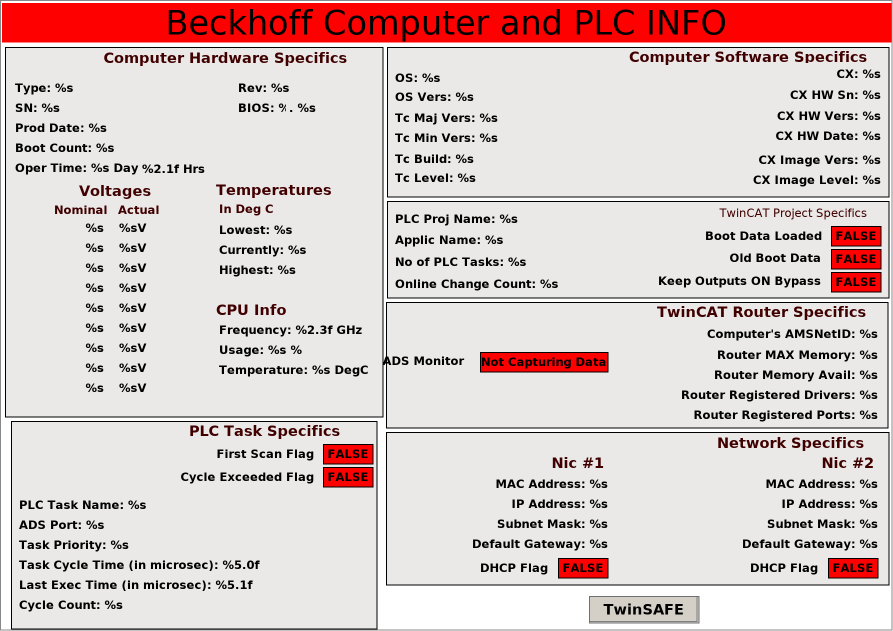
VISUALIZATION TwinCAT_INFO  // 893x631
    Button (589,596 110x27), "TwinSAFE"
        OnMouseClick: change screen: TwinSAFE
    RoundedRectangle (2,3 889x39), "Beckhoff Computer and PLC INFO"
    RoundedRectangle (387,47 502x150)
    Label (614,44 256x26), "Computer Software Specifics"
    Rectangle (392,67 256x22), "OS: %s", text variable: g_stHMI_DevIdent.strImageOsName
    RoundedRectangle (387,201 502x97)
    Label (695,200 175x26), "TwinCAT Project Specifics"
    RoundedRectangle (386,302 502x126)
    Label (613,299 256x26), "TwinCAT Router Specifics"
    RoundedRectangle (11,421 366x208)
    Label (185,418 158x26), "PLC Task Specifics"
    Rectangle (392,86 208x22), "OS Vers: %s", text variable: g_stHMI_DevIdent.strImageOsVersion
    Rectangle (392,107 119x22), "Tc Maj Vers: %s", text variable: g_stHMI_DevIdent.strTwinCATVersion
    Rectangle (392,127 111x22), "Tc Min Vers: %s", text variable: g_stHMI_DevIdent.strTwinCATRevision
    Rectangle (392,148 111x22), "Tc Build: %s", text variable: g_stHMI_DevIdent.strTwinCATBuild
    Rectangle (392,167 111x22), "Tc Level: %s", text variable: g_stHMI_DevIdent.strTwinCATLevel
    Rectangle (738,63 146x22), "CX: %s", text variable: g_stHMI_DevIdent.strHardwareModel
    Rectangle (726,84 158x22), "CX HW Sn: %s", text variable: g_stHMI_DevIdent.strHardwareSerialNo
    Rectangle (733,105 151x22), "CX HW Vers: %s", text variable: g_stHMI_DevIdent.strHardwareVersion
    Rectangle (737,125 147x22), "CX HW Date: %s", text variable: g_stHMI_DevIdent.strHardwareDate
    Rectangle (725,149 159x22), "CX Image Vers: %s", text variable: g_stHMI_DevIdent.strImageVersion
    Rectangle (625,169 259x22), "CX Image Level: %s", text variable: g_stHMI_DevIdent.strImageLevel
    Rectangle (392,208 283x22), "PLC Proj Name: %s", text variable: g_stHMI_AppInfo.ProjectName
    Rectangle (392,229 359x22), "Applic Name: %s", text variable: g_stHMI_AppInfo.AppName
    Rectangle (392,251 155x22), "No of PLC Tasks: %s", text variable: g_stHMI_AppInfo.TaskCnt
    Rectangle (392,273 191x22), "Online Change Count: %s", text variable: g_stHMI_AppInfo.OnlineChangeCnt
    Group (831,226 50x20)
        Rectangle (0,0 50x20), "TRUE", invisible if: NOT g_stHMI_AppInfo.BootDataLoaded
        Rectangle (0,0 50x20), "FALSE", invisible if: g_stHMI_AppInfo.BootDataLoaded
    Label (705,224 120x24), "Boot Data Loaded"
    Group (831,249 50x20)
        Rectangle (0,0 50x20), "TRUE", invisible if: NOT g_stHMI_AppInfo.OldBootData
        Rectangle (0,0 50x20), "FALSE", invisible if: g_stHMI_AppInfo.OldBootData
    Label (726,246 98x24), "Old Boot Data"
    Group (831,272 50x20)
        Rectangle (0,0 50x20), "TRUE", invisible if: NOT g_stHMI_AppInfo.KeepOutputsOnBP
        Rectangle (0,0 50x20), "FALSE", invisible if: NOT g_stHMI_AppInfo.KeepOutputsOnBP
    Label (682,269 142x24), "Keep Outputs ON Bypass"
    Label (392,349 75x24), "ADS Monitor"
    Group (480,352 128x20)
        Rectangle (0,0 128x20), "Capturing Data", invisible if: NOT g_stHMI_RouterStatusInfo.amsDebugLog
        Rectangle (0,0 128x20), "Not Capturing Data", invisible if: g_stHMI_RouterStatusInfo.amsDebugLog
    Rectangle (560,323 321x22), "Computer's AMSNetID: %s", text variable: g_stHMI_DevIdent.strAmsNetId
    Rectangle (673,344 208x22), "Router MAX Memory: %s", text variable: g_stHMI_RouterStatusInfo.maxMem
    Rectangle (673,364 208x22), "Router Memory Avail: %s", text variable: g_stHMI_RouterStatusInfo.maxMemAvail
    Rectangle (673,384 208x22), "Router Registered Drivers: %s", text variable: g_stHMI_RouterStatusInfo.regDrivers
    Rectangle (673,404 208x22), "Router Registered Ports: %s", text variable: g_stHMI_RouterStatusInfo.regPorts
    RoundedRectangle (5,47 378x370)
    Label (94,45 256x26), "Computer Hardware Specifics"
    Rectangle (12,77 141x22), "Type: %s", text variable: g_sHMI_MainboardType
    Rectangle (12,97 171x22), "SN: %s", text variable: g_sHMI_MainboardSN
    Rectangle (12,117 207x22), "Prod Date: %s", text variable: g_sHMI_MainboardProdDate
    Rectangle (12,137 151x22), "Boot Count: %s", text variable: g_udiHMI_MainboardBootCount
    Rectangle (12,157 184x22), "Oper Time: %s Days", text variable: g_udiHMI_MainboardOperTimeDays
    Rectangle (139,158 70x22), "%2.1f Hrs", text variable: g_lrHMI_MainboardOperTimeHrs
    Label (213,177 120x26), "Temperatures"
    Rectangle (216,219 102x22), "Lowest: %s", text variable: g_diHMI_MainboardMinTemp
    Rectangle (216,239 102x22), "Currently: %s", text variable: g_iHMI_MainboardActualTemp
    Rectangle (216,259 102x22), "Highest: %s", text variable: g_diHMI_MainboardMaxTemp
    Rectangle (235,77 67x22), "Rev: %s", text variable: g_bHMI_MainboardRevision
    Rectangle (235,97 67x22), "BIOS: %s", text variable: g_bHMI_MainboardBiosMajVers
    Rectangle (286,97 67x22), ". %s", text variable: g_bHMI_MainboardBiosMinVers
    Label (51,197 76x26), "Nominal"
    Rectangle (37,217 70x22), "%s", text variable: g_sHMI_Mainboard1p05v
    Rectangle (37,237 70x22), "%s", text variable: g_sHMI_MainboardVccCore
    Rectangle (37,257 70x22), "%s", text variable: g_sHMI_Mainboard5v
    Rectangle (37,277 70x22), "%s", text variable: g_sHMI_Mainboard12v
    Rectangle (37,297 70x22), "%s", text variable: g_sHMI_MainboardVBatt
    Rectangle (16,317 91x22), "%s", text variable: g_sHMI_MainboardPwrCtrlVcc
    Rectangle (16,337 91x22), "%s", text variable: g_sHMI_MainboardCX2100_5v
    Rectangle (18,357 89x22), "%s", text variable: g_sHMI_MainboardCX2100_12v
    Rectangle (19,377 88x22), "%s", text variable: g_sHMI_MainboardCX2100_24v
    Label (115,197 76x26), "Actual"
    Rectangle (116,217 70x22), "%sV", text variable: g_lrHMI_Mainboard1p05v
    Rectangle (116,237 70x22), "%sV", text variable: g_lrHMI_MainboardVccCore
    Rectangle (116,257 70x22), "%sV", text variable: g_lrHMI_Mainboard5v
    Rectangle (116,277 70x22), "%sV", text variable: g_lrHMI_Mainboard12v
    Rectangle (116,297 70x22), "%sV", text variable: g_lrHMI_MainboardVBatt
    Rectangle (116,317 91x22), "%sV", text variable: g_lrHMI_MainboardPwrCtrlVcc
    Rectangle (116,337 91x22), "%sV", text variable: g_lrHMI_MainboardCX2100_5v
    Rectangle (116,357 89x22), "%sV", text variable: g_lrHMI_MainboardCX2100_12v
    Rectangle (116,377 88x22), "%sV", text variable: g_lrHMI_MainboardCX2100_24v
    Label (76,178 71x26), "Voltages"
    Label (216,196 120x26), "In Deg C"
    Group (323,444 50x20)
        Rectangle (0,0 50x20), "TRUE", invisible if: NOT g_stHMI_PlcTaskSystemInfo.FirstCycle
        Rectangle (0,0 50x20), "FALSE", invisible if: g_stHMI_PlcTaskSystemInfo.FirstCycle
    Label (197,442 120x24), "First Scan Flag"
    Group (323,467 50x20)
        Rectangle (0,0 50x20), "TRUE", invisible if: NOT g_stHMI_PlcTaskSystemInfo.CycleTimeExceeded
        Rectangle (0,0 50x20), "FALSE", invisible if: g_stHMI_PlcTaskSystemInfo.CycleTimeExceeded
    Label (197,465 120x24), "Cycle Exceeded Flag"
    Rectangle (16,494 357x22), "PLC Task Name: %s", text variable: g_stHMI_PlcTaskSystemInfo.TaskName
    Rectangle (16,514 299x22), "ADS Port: %s", text variable: g_stHMI_PlcTaskSystemInfo.AdsPort
    Rectangle (16,534 214x22), "Task Priority: %s", text variable: g_stHMI_PlcTaskSystemInfo.Priority
    Rectangle (16,554 298x22), "Task Cycle Time (in microsec): %5.0f", text variable: g_lrHMI_PlcTaskSystemInfo_CycleTime
    Rectangle (16,574 298x22), "Last Exec Time (in microsec): %5.1f", text variable: g_lrHMI_PlcTaskSystemInfo_LastExecTime
    Rectangle (16,594 214x22), "Cycle Count: %s", text variable: g_stHMI_PlcTaskSystemInfo.CycleCount
    Label (213,297 120x26), "CPU Info"
    Rectangle (216,319 163x22), "Frequency: %2.3f GHz", text variable: g_lrHMI_CPUfrequency
    Rectangle (216,339 122x22), "Usage: %s %", text variable: g_iHMI_CPUusage
    Rectangle (216,359 156x22), "Temperature: %s DegC", text variable: g_iHMI_CPUtemperature
    RoundedRectangle (386,432 503x153)
    Label (716,430 151x26), "Network Specifics"
    Rectangle (396,473 215x22), "MAC Address: %s", text variable: System_Functions.ST_NIC0_ModContent.sMACAddress
    Rectangle (398,493 213x22), "IP Address: %s", text variable: System_Functions.ST_NIC0_ModContent.sIPAddress
    Rectangle (400,513 211x22), "Subnet Mask: %s", text variable: System_Functions.ST_NIC0_ModContent.sSubnetMask
    Rectangle (403,533 208x22), "Default Gateway: %s", text variable: System_Functions.ST_NIC0_ModContent.sDefaultGateway
    Group (558,558 50x20)
        Rectangle (0,0 50x20), "TRUE", invisible if: NOT System_Functions.ST_NIC0_ModContent.xDHCP
        Rectangle (0,0 50x20), "FALSE", invisible if: System_Functions.ST_NIC0_ModContent.xDHCP
    Label (481,556 70x24), "DHCP Flag"
    Label (456,450 151x26), "Nic #1"
    Rectangle (666,473 215x22), "MAC Address: %s", text variable: System_Functions.ST_NIC1_ModContent.sMACAddress
    Rectangle (668,493 213x22), "IP Address: %s", text variable: System_Functions.ST_NIC1_ModContent.sIPAddress
    Rectangle (670,513 211x22), "Subnet Mask: %s", text variable: System_Functions.ST_NIC1_ModContent.sSubnetMask
    Rectangle (673,533 208x22), "Default Gateway: %s", text variable: System_Functions.ST_NIC1_ModContent.sDefaultGateway
    Group (828,558 50x20)
        Rectangle (0,0 50x20), "TRUE", invisible if: NOT System_Functions.ST_NIC1_ModContent.xDHCP
        Rectangle (0,0 50x20), "FALSE", invisible if: System_Functions.ST_NIC1_ModContent.xDHCP
    Label (751,556 70x24), "DHCP Flag"
    Label (726,450 151x26), "Nic #2"
END_VISUALIZATION

(* stored: Version 1.1.0.1, ProductVersion 3.1.0.18
   Visu TwinCAT_INFO: Id {319d32cd-6358-4f17-a08d-5447f8085241} *)
